RoboDK station: V2_FeedingProject_Assistive_UR5e.rdk

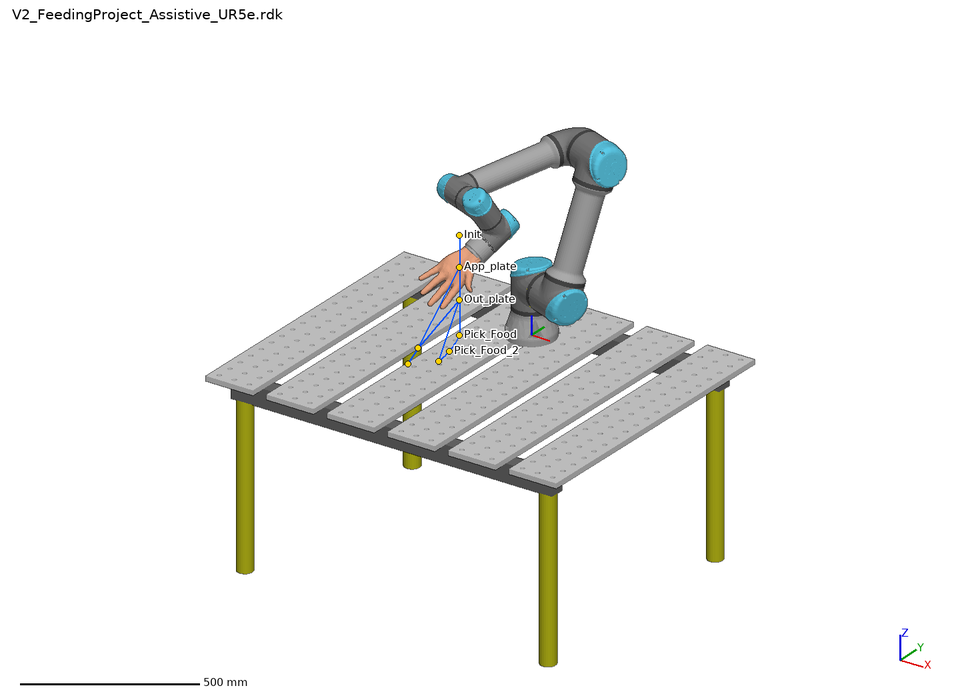
[picture v0: the station drawn from its stored meshes, robots at their saved joint values, targets as dots, program paths as lines]
Station V2_FeedingProject_Assistive_UR5e (saved by RoboDK 5.9.2). Poses are relative to the parent item; angles as X-Y-Z fixed-axis rotations.
  - frame UR5e Base at (0, 0, 0) mm
    - robot UR5e: 6 axes, payload 5 kg, reach 850 mm, repeatability 0.03 mm, weight 18.4 kg
        modified DH rows (alpha deg, a mm, theta deg, d mm): 0, 0, 0, 162.5; 90, 0, 180, 0; 0, 425, 0, 0; 0, 392.25, 0, 133.3; -90, 0, 0, 99.7; 90, 0, 180, 99.6
        joint limits [-360, -360, -360, -360, -360, -360] to [360, 360, 360, 360, 360, 360]; home [0, -90, -90, 0, 90, 0]; saved at [68.192, -108.662, 116.049, 25.329, -268.745, 248.075]
      - tool Hand, TCP at (0, 0, 50) mm, size 54.8 x 155.9 x 193.5 mm, geometry from Hand.stl
  - frame World at (0, 0, 0) mm
    - object Table at (0, 0, 0) mm, size 1193.8 x 965.2 x 609.6 mm, geometry from welding_table.sld
    - target Init (Cartesian target) at (0, -350, 450) mm, rotated rx -148.96 ry 50.9 rz 104.49 deg; joints [68.193, -108.676, 101.412, 39.982, -268.742, 248.077] of UR5e
    - target App_plate (Cartesian target) at (0, -350, 350) mm, rotated rx -148.96 ry 50.9 rz 104.49 deg; joints [68.192, -108.662, 116.049, 25.329, -268.745, 248.075] of UR5e
    - target Pick_Food (Cartesian target) at (0, -350, 140) mm, rotated rx 134.4 ry 73.3 rz 17.94 deg; joints [69.922, -93.417, 147.836, -42.773, -264.959, 283.136] of UR5e
    - target Pick_Food_2 (Cartesian target) at (0, -400, 110) mm, rotated rx 134.4 ry 73.3 rz 17.94 deg; joints [74.107, -80.317, 141.524, -49.455, -260.861, 283.991] of UR5e
    - target Pick_Food_3 (Cartesian target) at (0, -450, 100) mm, rotated rx 134.4 ry 73.3 rz 17.94 deg; joints [76.798, -73.218, 133.82, -48.75, -258.227, 284.551] of UR5e
    - target Out_plate (Cartesian target) at (0, -350, 250) mm, rotated rx 134.4 ry 73.3 rz 17.94 deg; joints [69.922, -109.66, 137.8, -16.494, -264.959, 283.136] of UR5e
    - target App_mouth (Cartesian target) at (0, -550, 180) mm, rotated rx 134.4 ry 73.3 rz 17.94 deg; joints [80.099, -72.507, 114.073, -29.55, -254.997, 285.252] of UR5e
    - target In_mouth (Cartesian target) at (0, -600, 150) mm, rotated rx 134.4 ry 73.3 rz 17.94 deg; joints [81.191, -64.054, 106.97, -30.836, -253.929, 285.489] of UR5e
  - program Feeding (13 instructions, listed below)
  - program MainProgram (3 instructions, listed below)
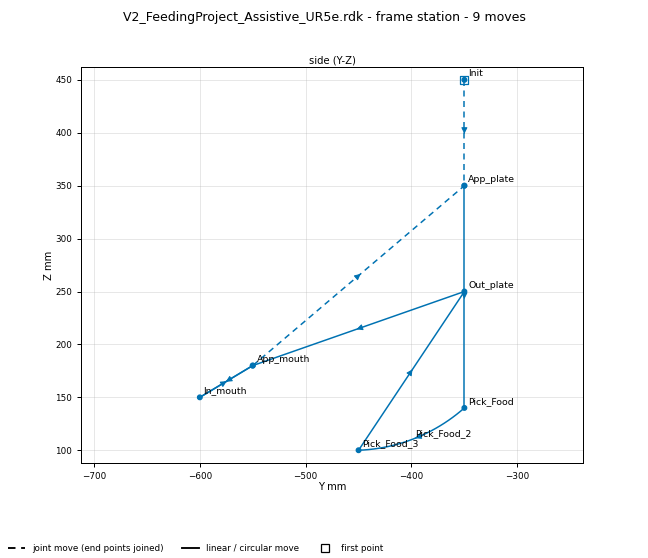
[picture p0: tool path of V2_FeedingProject_Assistive_UR5e.rdk in frame station, 9 of 9 moves have a stored position in this frame; points joined in program order, loops and branches not executed]

--- program Feeding (robot UR5e) ---
  Est. Ref.: UR5e Base
  Est. herr: Hand
  MoveJ (Init)
  MoveJ (App_plate)
  MoveL (Pick_Food)
  MoveC (Pick_Food_2, Pick_Food_3)
  Pausa 1.0 s
  MoveL (Out_plate)
  MoveL (App_mouth)
  MoveL (In_mouth)
  Pausa 3.0 s
  MoveL (App_mouth)
  MoveJ (App_plate)

--- program MainProgram (robot UR5e) ---
  Establecer velocidad (600.0 mm/s)
  Llamar Feeding
  Pausa 4.0 s
